PROGRAM pouMcPrompts
VAR
	


idbMsgPrompt: FB_CheckMessageBounds;
END_VAR

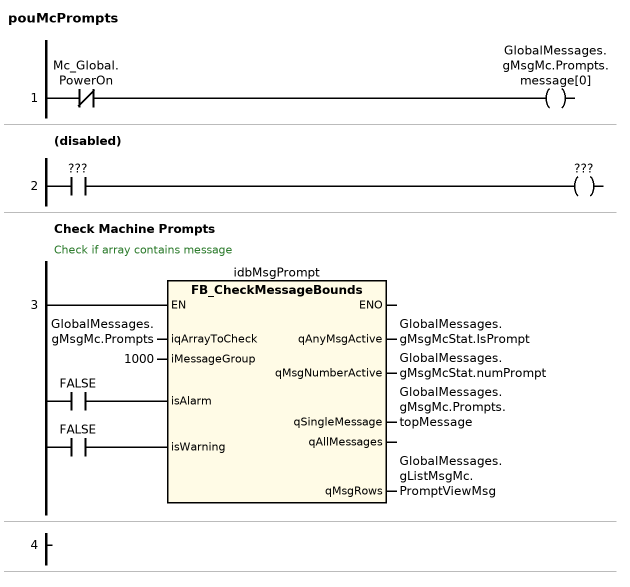
// NETWORK 1
GlobalMessages.gMsgMc.Prompts.message[0] := NOT Mc_Global.PowerOn;

// NETWORK 2 (disabled)
// ??? := ???;

// NETWORK 3: Check Machine Prompts
// Check if array contains message
idbMsgPrompt(
    iqArrayToCheck := GlobalMessages.gMsgMc.Prompts,
    iMessageGroup := 1000,
    isAlarm := FALSE,
    isWarning := FALSE,
    qAnyMsgActive => GlobalMessages.gMsgMcStat.IsPrompt,
    qMsgNumberActive => GlobalMessages.gMsgMcStat.numPrompt,
    qSingleMessage => GlobalMessages.gMsgMc.Prompts.topMessage,
    qMsgRows => GlobalMessages.gListMsgMc.PromptViewMsg); // FB_CheckMessageBounds

// NETWORK 4

END_PROGRAM

(* stored: Version 1.1.0.1, ProductVersion 3.1.4024.12
   POU pouMcPrompts: Id {d586c653-4092-490f-b1fa-a2659fd64310}, SpecialFunc None *)
